// TIA Portal V20 export
// export: Created 2025-12-01T14:57:11.2928145Z, ExportSetting None, DisplayName Totally Integrated Automation Portal, DisplayVersion V20 Update 3, DisplayName TIA Portal Openness, DisplayVersion V20 Update 3, DisplayName TIA Portal Version Control Interface, DisplayVersion V20 Update 3, DisplayName STEP 7 Professional, DisplayVersion V20 Update 3, DisplayName STEP 7 Safety, DisplayVersion V20 Update 2, DisplayName WinCC Basic/Comfort/Advanced, DisplayVersion V20 Update 3, DisplayName WinCC Professional, DisplayVersion V20 Update 3, DisplayName WinCC Unified, DisplayVersion V20 Update 3
FUNCTION "FC895_Obtener_EtiquetaDeValor" : Void   // FC895, LAD
TITLE = "Evento_ValorEtiqueta
{ S7_Optimized_Access := 'FALSE' }
AUTHOR : TRACKING
NAME : 20160407
VERSION : 3.3
// Convertir un valor numerico UInt a un texto DWORD
// stored: AutoNumber false, SetENOAutomatically false
   VAR_INPUT
      ValorEvento : UInt;   // Valor del Evento a Enviar
   END_VAR
   VAR_OUTPUT
      EtiquetaEvento : DWord;   // Etiqueta del Evento a Enviar
   END_VAR
   VAR_TEMP
      Indice : UInt;
   END_VAR
BEGIN

NETWORK
TITLE = Inicializar
// - Inicializar la salida de la función
      L     '----';
      T     #EtiquetaEvento;


NETWORK
TITLE = Buscar la Etiqueta
/////////////////////////////////////////////////////////////////////////////////////
/////////////////////////////////////////////////////////////////////////////////////
/////////////////////////////////////////////////////////////////////////////////////
// --- Bucle de Busqueda de Etiqueta
      L     1;
      T     #Indice;

Inicio_BucleDeBusqueda:NOP   0;
      L     "DB870_ConversorEventos".Valor_A_Etiqueta[#Indice].Valor;
      L     #ValorEvento;
      ==I;
      JC    Encontrada_EtiquetaBuscada;

// --- Final de Etiquetas Existentes
      L     "DB870_ConversorEventos".Valor_A_Etiqueta[#Indice].Valor;
      L     0;
      ==I;
      JC    Final;  // Hay mas etiquetas?

// --- Maximo del Array de Etiquetas
      L     #Indice;
      L     "CTE_MaxArrayConversion";
      >=I;
      JC    Final;  // No se ha encontrado?


// --- Continuar la Busqueda
      L     #Indice;
      L     1;
      +I;
      T     #Indice;

      JU    Inicio_BucleDeBusqueda;

/////////////////////////////////////////////////////////////////////////////////////
/////////////////////////////////////////////////////////////////////////////////////
/////////////////////////////////////////////////////////////////////////////////////
// --- Etiqueta Encontrada
Encontrada_EtiquetaBuscada:NOP   0;
      L     "DB870_ConversorEventos".Valor_A_Etiqueta[#Indice].Etiqueta;
      T     #EtiquetaEvento;



NETWORK
TITLE = Finalizar
/////////////////////////////////////////////////////////////////////////////////////
// Final de la funcion
Final:NOP   0;

END_FUNCTION
